// SIMATIC S7-200 project (STEP 7-Micro/WIN), CPU 224 AM REL 21.02

ORGANIZATION_BLOCK 主程序:OB1
TITLE=程序注释
BEGIN
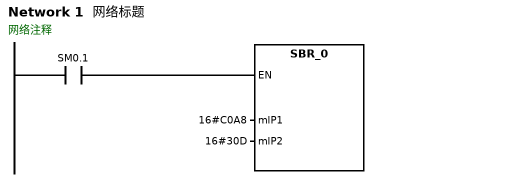
Network 1 // 网络标题
// 网络注释
LD     SM0.1
CALL   SBR_0:SBR0, 16#C0A8, 16#30D
END_ORGANIZATION_BLOCK

SUBROUTINE_BLOCK SBR_0:SBR0
TITLE=子程序注释
VAR_INPUT
mlP1:WORD;	// LW0 
mlP2:WORD;	// LW2 
END_VAR
BEGIN
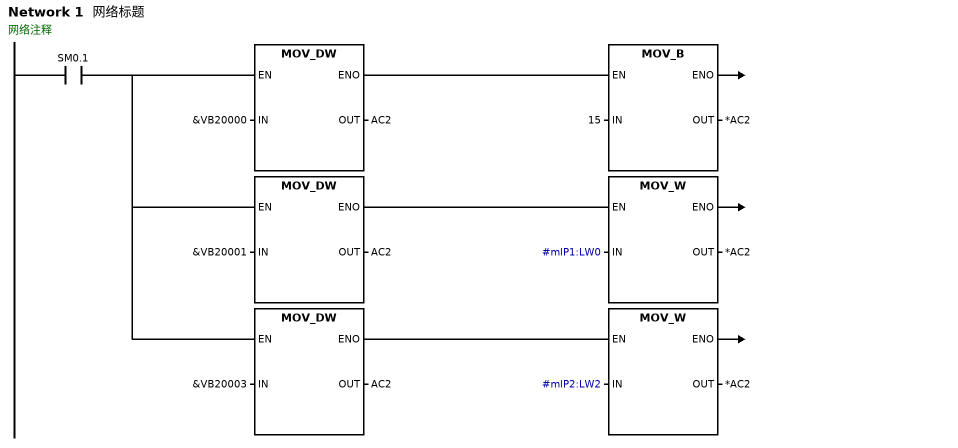
Network 1 // 网络标题
// 网络注释
LD     SM0.1
LPS
MOVD   &VB20000, AC2
AENO
MOVB   15, *AC2
LRD
MOVD   &VB20001, AC2
AENO
MOVW   #mlP1:LW0, *AC2
LPP
MOVD   &VB20003, AC2
AENO
MOVW   #mlP2:LW2, *AC2
END_SUBROUTINE_BLOCK
